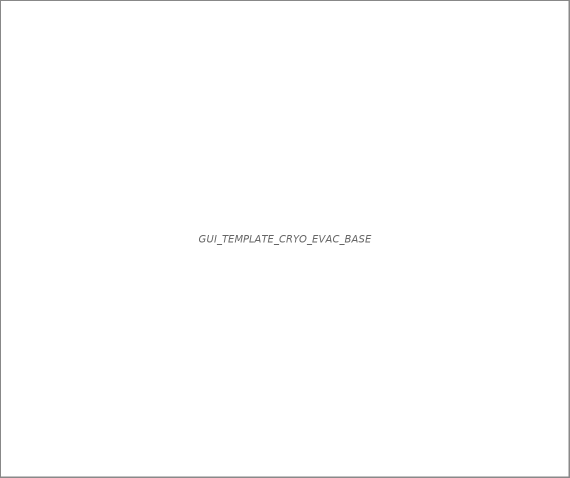
VISUALIZATION GUI_EVAC_PDS  // 570x478
    Frame (0,0 570x478)
        shows GUI_TEMPLATE_CRYO_EVAC_BASE(m_Instance := MAIN.evac_pds, m_bEnable := MAIN.bEnable_evac_pds)
END_VISUALIZATION

(* stored: Version 1.1.0.1, ProductVersion 3.1.4024.9
   Visu GUI_EVAC_PDS: Id {951bfc88-0ae6-4fee-aff6-2ddcdd7991be} *)
